Fanuc KAREL source: kx00026.KL

-- PROVISIONAL review KL for V770-1; original PC SHA256 fb05bdd3397013ca1b9ea2a4f4c0103d549d406c76c9d4cc1d67d57f2c8004e1
-- Incomplete behavior may be omitted. Consult companion uncertainty JSON. Do not deploy.
PROGRAM KX00026
%NOLOCKGROUP
VAR
  I : INTEGER
  J : INTEGER
  B : BOOLEAN
  F : FILE
  S : STRING[80]
-- UNRESOLVED_DECL P type=000102
BEGIN
  -- UNRESOLVED_PC offsets 5-12; opcodes 9D,23
  -- UNRESOLVED_PC offsets 17-21; opcodes 7F
END KX00026
